FUNCTION_BLOCK RingTokenNetworkTwo (* Composite Function Block Type *)
  (* Standard: 61499-2 *)
  (* Version 0.2, 2003-12-05, JHC, Rockwell Automation, Renamed from NEWCOMPFB. *)
  (* Version 0.1, 2002-01-08, JHC, Rockwell Automation, Added DLY FB as example. *)
  (* Version 0.0, 2000-05-27, JHC, Rockwell Automation *)
  (* Compiler header: package fb.rt.template; *)
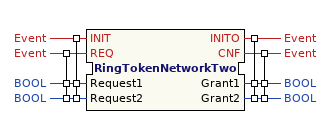
  EVENT_INPUT
    INIT WITH Request1, Request2; (* Initialization Request *)
    REQ WITH Request1, Request2; (* Normal Execution Request *)
  END_EVENT
  EVENT_OUTPUT
    INITO WITH Grant1, Grant2; (* Initialization Confirm *)
    CNF WITH Grant1, Grant2; (* Execution Confirmation *)
  END_EVENT
  VAR_INPUT
    Request1 : BOOL; (* Input event qualifier *)
    Request2 : BOOL;
  END_VAR
  VAR_OUTPUT
    Grant1 : BOOL; (* Output event qualifier *)
    Grant2 : BOOL;
  END_VAR
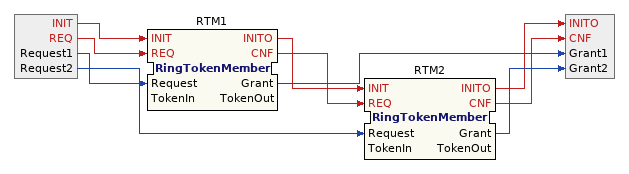
  FBS
    RTM1 : RingTokenMember;
    RTM2 : RingTokenMember;
  END_FBS
  EVENT_CONNECTIONS
    RTM1.INITO TO RTM2.INIT;
    INIT TO RTM1.INIT;
    RTM2.INITO TO INITO;
    RTM2.CNF TO CNF;
    REQ TO RTM1.REQ;
    RTM1.CNF TO RTM2.REQ;
  END_CONNECTIONS
  DATA_CONNECTIONS
    RTM1.Grant TO Grant1;
    RTM2.Grant TO Grant2;
    Request2 TO RTM2.Request;
    Request1 TO RTM1.Request;
  END_CONNECTIONS
END_FUNCTION_BLOCK
